(* PLC project CoDeSys External Library Template, WAGO e!COCKPIT e!COCKPIT, author 3S - Smart Software Solutions GmbH *)
(* stored: creationDateTime 2019-10-29T12:22:40.9579989, version 3.5.5.30, modificationDateTime 2019-10-24T14:40:07.960949, organization 3S - Smart Software Solutions GmbH *)
(* Library project template with all possible element types, docu and a sample project structure *)

FUNCTION fnKonwersjaINT_STRING : STRING
  VAR_INPUT
    intWartosc : INT;
    intIloscZnakow : INT;
  END_VAR

            fnKonwersjaINT_STRING := INT_TO_STRING(intWartosc);

IF intWartosc < 100000 AND intIloscZnakow > 5 THEN
	fnKonwersjaINT_STRING := CONCAT('0' , fnKonwersjaINT_STRING);
END_IF

IF intWartosc < 10000 AND intIloscZnakow > 4 THEN
	fnKonwersjaINT_STRING := CONCAT('0' , fnKonwersjaINT_STRING);
END_IF

IF intWartosc < 1000 AND intIloscZnakow > 3 THEN
	fnKonwersjaINT_STRING := CONCAT('0' , fnKonwersjaINT_STRING);
END_IF

IF intWartosc < 100 AND intIloscZnakow > 2 THEN
	fnKonwersjaINT_STRING := CONCAT('0' , fnKonwersjaINT_STRING);
END_IF

IF intWartosc < 10 AND intIloscZnakow > 1 THEN
	fnKonwersjaINT_STRING := CONCAT('0' , fnKonwersjaINT_STRING);
END_IF

          
END_FUNCTION
